FUNCTION_BLOCK TestBitAdrState EXTENDS TcUnit.FB_TestSuite
VAR_INPUT
END_VAR
VAR_OUTPUT
END_VAR
VAR
END_VAR

first_bit_of_first_byte_is_off();
first_bit_of_first_byte_is_on();
last_bit_of_first_byte_is_off();
last_bit_of_first_byte_is_on();
first_bit_of_second_byte_is_off();
first_bit_of_second_byte_is_on();
last_bit_of_second_byte_is_off();
last_bit_of_second_byte_is_on();
fourth_bit_of_second_byte_is_on();
negative_bit_adr_is_off();
out_of_bounds_bit_adr_is_off();

METHOD first_bit_of_first_byte_is_off
VAR
  state: BOOL;
END_VAR
VAR_INST
  b: ARRAY[0..1] OF BYTE;
END_VAR
TEST('first_bit_of_first_byte_is_off');

state := BitAdrState(0, ADR(b), SIZEOF(b));
AssertFalse(state, '');

TEST_FINISHED();
END_METHOD

METHOD last_bit_of_second_byte_is_off
VAR
  state: BOOL;
END_VAR
VAR_INST
  b: ARRAY[0..1] OF BYTE;
END_VAR
TEST('last_bit_of_second_byte_is_off');

b[1] := 0;
state := BitAdrState(15, ADR(b), SIZEOF(b));
AssertFalse(state, '');

TEST_FINISHED();
END_METHOD

METHOD last_bit_of_first_byte_is_on
VAR
  state: BOOL;
END_VAR
VAR_INST
  b: ARRAY[0..1] OF BYTE;
END_VAR
TEST('last_bit_of_first_byte_is_on');

b[0] := 128;
state := BitAdrState(7, ADR(b), SIZEOF(b));
AssertTrue(state, '');

TEST_FINISHED();
END_METHOD

METHOD first_bit_of_second_byte_is_on
VAR
  state: BOOL;
END_VAR
VAR_INST
  b: ARRAY[0..1] OF BYTE;
END_VAR
TEST('first_bit_of_second_byte_is_on');

b[1] := 1;
state := BitAdrState(8, ADR(b), SIZEOF(b));
AssertTrue(state, '');

TEST_FINISHED();
END_METHOD

METHOD first_bit_of_first_byte_is_on
VAR
  state: BOOL;
END_VAR
VAR_INST
  b: ARRAY[0..1] OF BYTE;
END_VAR
TEST('first_bit_of_first_byte_is_on');

b[0] := 1;
state := BitAdrState(0, ADR(b), SIZEOF(b));
AssertTrue(state, '');

TEST_FINISHED();
END_METHOD

METHOD first_bit_of_second_byte_is_off
VAR
  state: BOOL;
END_VAR
VAR_INST
  b: ARRAY[0..1] OF BYTE;
END_VAR
TEST('first_bit_of_second_byte_is_off');

b[1] := 0;
state := BitAdrState(8, ADR(b), SIZEOF(b));
AssertFalse(state, '');

TEST_FINISHED();
END_METHOD

METHOD fourth_bit_of_second_byte_is_on
VAR
  state: BOOL;
END_VAR
VAR_INST
  b: ARRAY[0..1] OF BYTE;
END_VAR
TEST('fourth_bit_of_second_byte_is_on');

b[1] := 8;
state := BitAdrState(11, ADR(b), SIZEOF(b));
AssertTrue(state, '');

TEST_FINISHED();
END_METHOD

METHOD last_bit_of_first_byte_is_off
VAR
  state: BOOL;
END_VAR
VAR_INST
  b: ARRAY[0..1] OF BYTE;
END_VAR
TEST('last_bit_of_first_byte_is_off');

b[0] := 0;
state := BitAdrState(7, ADR(b), SIZEOF(b));
AssertFalse(state, '');

TEST_FINISHED();
END_METHOD

METHOD out_of_bounds_bit_adr_is_off
VAR
  state: BOOL;
END_VAR
VAR_INST
  b: ARRAY[0..1] OF BYTE;
END_VAR
TEST('out_of_bounds_bit_adr_is_off');

b[0] := 255;
b[1] := 255;
state := BitAdrState(16, ADR(b), SIZEOF(b));
AssertFalse(state, '');

TEST_FINISHED();
END_METHOD

METHOD last_bit_of_second_byte_is_on
VAR
  state: BOOL;
END_VAR
VAR_INST
  b: ARRAY[0..1] OF BYTE;
END_VAR
TEST('last_bit_of_second_byte_is_on');

b[1] := 128;
state := BitAdrState(15, ADR(b), SIZEOF(b));
AssertTrue(state, '');

TEST_FINISHED();
END_METHOD

METHOD negative_bit_adr_is_off
VAR
  state: BOOL;
END_VAR
VAR_INST
  b: ARRAY[0..1] OF BYTE;
END_VAR
TEST('negative_bit_adr_is_off');

b[0] := 1;
state := BitAdrState(-1, ADR(b), SIZEOF(b));
AssertFalse(state, '');

TEST_FINISHED();
END_METHOD

END_FUNCTION_BLOCK

(* stored: Version 1.1.0.1, ProductVersion 3.1.4022.18
   POU TestBitAdrState: Id {547edaea-38e9-474b-af76-454c809a918a}, SpecialFunc None
   Method first_bit_of_first_byte_is_off: Id {0e64da5e-3594-4252-93eb-f5145e0d8470}
   Method last_bit_of_second_byte_is_off: Id {302c403d-a6cf-4137-bfbe-284f1bc1be54}
   Method last_bit_of_first_byte_is_on: Id {4792c87b-119a-451d-b5eb-041f0db8233e}
   Method first_bit_of_second_byte_is_on: Id {4c5c9b74-9114-4f2e-9ee3-07371a5227c9}
   Method first_bit_of_first_byte_is_on: Id {503208ef-f957-426d-a272-d396a3639452}
   Method first_bit_of_second_byte_is_off: Id {60105bd8-0dab-46b8-9e41-8ae200f07c27}
   Method fourth_bit_of_second_byte_is_on: Id {a25d06ce-ed52-4cbd-8130-02c75e84d22d}
   Method last_bit_of_first_byte_is_off: Id {a6898c4a-b727-4125-84f4-baaab049d4f6}
   Method out_of_bounds_bit_adr_is_off: Id {d518ca4e-f9ef-4f37-9d06-fe80d7e35a0f}
   Method last_bit_of_second_byte_is_on: Id {e71c92ac-5bf8-4df3-b721-199595454953}
   Method negative_bit_adr_is_off: Id {f128680f-e3f2-43b9-a8bf-f2d24073c69e} *)
